FUNCTION SPLITTING_LWORD_INTO_BOOLS
  (* Standard: 61499-1; Description: Copyright (c) 2024 HR Agrartechnik GmbH This program and the accompanying materials are made available under the terms of the Eclipse Public License 2.0 which is available at https://www.eclipse.org/legal/epl-2.0/ SPDX-License-Identifier: EPL-2.0 *)
  (* Version 1.0, 2024-02-22, franz *)
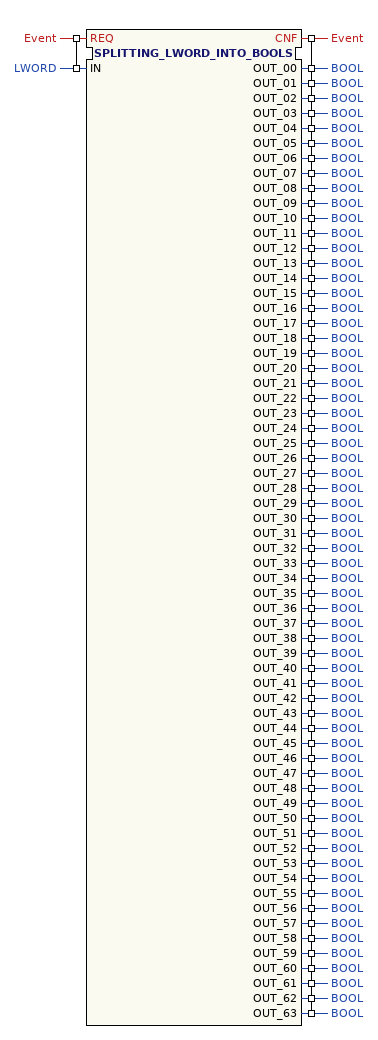
  EVENT_INPUT
    REQ WITH IN; (* Normal Execution Request *)
  END_EVENT
  EVENT_OUTPUT
    CNF WITH OUT_00, OUT_01, OUT_02, OUT_03, OUT_04, OUT_05, OUT_06, OUT_07, OUT_08, OUT_09, OUT_10, OUT_11, OUT_12, OUT_13, OUT_14, OUT_15, OUT_16, OUT_17, OUT_18, OUT_19, OUT_20, OUT_21, OUT_22, OUT_23, OUT_24, OUT_25, OUT_26, OUT_27, OUT_28, OUT_29, OUT_30, OUT_31, OUT_32, OUT_33, OUT_34, OUT_35, OUT_36, OUT_37, OUT_38, OUT_39, OUT_40, OUT_41, OUT_42, OUT_43, OUT_44, OUT_45, OUT_46, OUT_47, OUT_48, OUT_49, OUT_50, OUT_51, OUT_52, OUT_53, OUT_54, OUT_55, OUT_56, OUT_57, OUT_58, OUT_59, OUT_60, OUT_61, OUT_62, OUT_63; (* Execution Confirmation *)
  END_EVENT
  VAR_INPUT
    IN : LWORD; (* LWORD Input *)
  END_VAR
  VAR_OUTPUT
    OUT_00 : BOOL; (* BIT 00 *)
    OUT_01 : BOOL; (* BIT 01 *)
    OUT_02 : BOOL; (* BIT 02 *)
    OUT_03 : BOOL; (* BIT 03 *)
    OUT_04 : BOOL; (* BIT 04 *)
    OUT_05 : BOOL; (* BIT 05 *)
    OUT_06 : BOOL; (* BIT 06 *)
    OUT_07 : BOOL; (* BIT 07 *)
    OUT_08 : BOOL; (* BIT 08 *)
    OUT_09 : BOOL; (* BIT 09 *)
    OUT_10 : BOOL; (* BIT 10 *)
    OUT_11 : BOOL; (* BIT 11 *)
    OUT_12 : BOOL; (* BIT 12 *)
    OUT_13 : BOOL; (* BIT 13 *)
    OUT_14 : BOOL; (* BIT 14 *)
    OUT_15 : BOOL; (* BIT 15 *)
    OUT_16 : BOOL; (* BIT 16 *)
    OUT_17 : BOOL; (* BIT 17 *)
    OUT_18 : BOOL; (* BIT 18 *)
    OUT_19 : BOOL; (* BIT 19 *)
    OUT_20 : BOOL; (* BIT 20 *)
    OUT_21 : BOOL; (* BIT 21 *)
    OUT_22 : BOOL; (* BIT 22 *)
    OUT_23 : BOOL; (* BIT 23 *)
    OUT_24 : BOOL; (* BIT 24 *)
    OUT_25 : BOOL; (* BIT 25 *)
    OUT_26 : BOOL; (* BIT 26 *)
    OUT_27 : BOOL; (* BIT 27 *)
    OUT_28 : BOOL; (* BIT 28 *)
    OUT_29 : BOOL; (* BIT 29 *)
    OUT_30 : BOOL; (* BIT 30 *)
    OUT_31 : BOOL; (* BIT 31 *)
    OUT_32 : BOOL; (* BIT 32 *)
    OUT_33 : BOOL; (* BIT 33 *)
    OUT_34 : BOOL; (* BIT 34 *)
    OUT_35 : BOOL; (* BIT 35 *)
    OUT_36 : BOOL; (* BIT 36 *)
    OUT_37 : BOOL; (* BIT 37 *)
    OUT_38 : BOOL; (* BIT 38 *)
    OUT_39 : BOOL; (* BIT 39 *)
    OUT_40 : BOOL; (* BIT 40 *)
    OUT_41 : BOOL; (* BIT 41 *)
    OUT_42 : BOOL; (* BIT 42 *)
    OUT_43 : BOOL; (* BIT 43 *)
    OUT_44 : BOOL; (* BIT 44 *)
    OUT_45 : BOOL; (* BIT 45 *)
    OUT_46 : BOOL; (* BIT 46 *)
    OUT_47 : BOOL; (* BIT 47 *)
    OUT_48 : BOOL; (* BIT 48 *)
    OUT_49 : BOOL; (* BIT 49 *)
    OUT_50 : BOOL; (* BIT 50 *)
    OUT_51 : BOOL; (* BIT 51 *)
    OUT_52 : BOOL; (* BIT 52 *)
    OUT_53 : BOOL; (* BIT 53 *)
    OUT_54 : BOOL; (* BIT 54 *)
    OUT_55 : BOOL; (* BIT 55 *)
    OUT_56 : BOOL; (* BIT 56 *)
    OUT_57 : BOOL; (* BIT 57 *)
    OUT_58 : BOOL; (* BIT 58 *)
    OUT_59 : BOOL; (* BIT 59 *)
    OUT_60 : BOOL; (* BIT 60 *)
    OUT_61 : BOOL; (* BIT 61 *)
    OUT_62 : BOOL; (* BIT 62 *)
    OUT_63 : BOOL; (* BIT 63 *)
  END_VAR
  BODY IN ST:
FUNCTION SPLITTING_LWORD_INTO_BOOLS

VAR_INPUT
	IN : LWORD;    // LWORD Input
END_VAR

VAR_OUTPUT
	OUT_00 : BOOL;    // BIT 00
	OUT_01 : BOOL;    // BIT 01
	OUT_02 : BOOL;    // BIT 02
	OUT_03 : BOOL;    // BIT 03
	OUT_04 : BOOL;    // BIT 04
	OUT_05 : BOOL;    // BIT 05
	OUT_06 : BOOL;    // BIT 06
	OUT_07 : BOOL;    // BIT 07
	OUT_08 : BOOL;    // BIT 08
	OUT_09 : BOOL;    // BIT 09
	OUT_10 : BOOL;    // BIT 10
	OUT_11 : BOOL;    // BIT 11
	OUT_12 : BOOL;    // BIT 12
	OUT_13 : BOOL;    // BIT 13
	OUT_14 : BOOL;    // BIT 14
	OUT_15 : BOOL;    // BIT 15
	OUT_16 : BOOL;    // BIT 16
	OUT_17 : BOOL;    // BIT 17
	OUT_18 : BOOL;    // BIT 18
	OUT_19 : BOOL;    // BIT 19
	OUT_20 : BOOL;    // BIT 20
	OUT_21 : BOOL;    // BIT 21
	OUT_22 : BOOL;    // BIT 22
	OUT_23 : BOOL;    // BIT 23
	OUT_24 : BOOL;    // BIT 24
	OUT_25 : BOOL;    // BIT 25
	OUT_26 : BOOL;    // BIT 26
	OUT_27 : BOOL;    // BIT 27
	OUT_28 : BOOL;    // BIT 28
	OUT_29 : BOOL;    // BIT 29
	OUT_30 : BOOL;    // BIT 30
	OUT_31 : BOOL;    // BIT 31
	OUT_32 : BOOL;    // BIT 32
	OUT_33 : BOOL;    // BIT 33
	OUT_34 : BOOL;    // BIT 34
	OUT_35 : BOOL;    // BIT 35
	OUT_36 : BOOL;    // BIT 36
	OUT_37 : BOOL;    // BIT 37
	OUT_38 : BOOL;    // BIT 38
	OUT_39 : BOOL;    // BIT 39
	OUT_40 : BOOL;    // BIT 40
	OUT_41 : BOOL;    // BIT 41
	OUT_42 : BOOL;    // BIT 42
	OUT_43 : BOOL;    // BIT 43
	OUT_44 : BOOL;    // BIT 44
	OUT_45 : BOOL;    // BIT 45
	OUT_46 : BOOL;    // BIT 46
	OUT_47 : BOOL;    // BIT 47
	OUT_48 : BOOL;    // BIT 48
	OUT_49 : BOOL;    // BIT 49
	OUT_50 : BOOL;    // BIT 50
	OUT_51 : BOOL;    // BIT 51
	OUT_52 : BOOL;    // BIT 52
	OUT_53 : BOOL;    // BIT 53
	OUT_54 : BOOL;    // BIT 54
	OUT_55 : BOOL;    // BIT 55
	OUT_56 : BOOL;    // BIT 56
	OUT_57 : BOOL;    // BIT 57
	OUT_58 : BOOL;    // BIT 58
	OUT_59 : BOOL;    // BIT 59
	OUT_60 : BOOL;    // BIT 60
	OUT_61 : BOOL;    // BIT 61
	OUT_62 : BOOL;    // BIT 62
	OUT_63 : BOOL;    // BIT 63
END_VAR

(* this Function extracts the 64 BOOLS from a lword *)
OUT_00 := IN.0;
OUT_01 := IN.1;
OUT_02 := IN.2;
OUT_03 := IN.3;
OUT_04 := IN.4;
OUT_05 := IN.5;
OUT_06 := IN.6;
OUT_07 := IN.7;
OUT_08 := IN.8;
OUT_09 := IN.9;
OUT_10 := IN.10;
OUT_11 := IN.11;
OUT_12 := IN.12;
OUT_13 := IN.13;
OUT_14 := IN.14;
OUT_15 := IN.15;
OUT_16 := IN.16;
OUT_17 := IN.17;
OUT_18 := IN.18;
OUT_19 := IN.19;
OUT_20 := IN.20;
OUT_21 := IN.21;
OUT_22 := IN.22;
OUT_23 := IN.23;
OUT_24 := IN.24;
OUT_25 := IN.25;
OUT_26 := IN.26;
OUT_27 := IN.27;
OUT_28 := IN.28;
OUT_29 := IN.29;
OUT_30 := IN.30;
OUT_31 := IN.31;
OUT_32 := IN.32;
OUT_33 := IN.33;
OUT_34 := IN.34;
OUT_35 := IN.35;
OUT_36 := IN.36;
OUT_37 := IN.37;
OUT_38 := IN.38;
OUT_39 := IN.39;
OUT_40 := IN.40;
OUT_41 := IN.41;
OUT_42 := IN.42;
OUT_43 := IN.43;
OUT_44 := IN.44;
OUT_45 := IN.45;
OUT_46 := IN.46;
OUT_47 := IN.47;
OUT_48 := IN.48;
OUT_49 := IN.49;
OUT_50 := IN.50;
OUT_51 := IN.51;
OUT_52 := IN.52;
OUT_53 := IN.53;
OUT_54 := IN.54;
OUT_55 := IN.55;
OUT_56 := IN.56;
OUT_57 := IN.57;
OUT_58 := IN.58;
OUT_59 := IN.59;
OUT_60 := IN.60;
OUT_61 := IN.61;
OUT_62 := IN.62;
OUT_63 := IN.63;
END_FUNCTION
  END_BODY
END_FUNCTION
